TYPE ST_MyData :
STRUCT
	Nr		: DINT;
	Zeit 	: DT;
	Wert 	: REAL;
END_STRUCT
END_TYPE

(* stored: Version 1.1.0.1
   DUT ST_MyData: Id {2287a124-1aca-471e-beef-441c47bddcd9} *)
